// TIA Portal V17 export
// export: Created 2025-06-25T13:13:26.438801Z, ExportSetting WithDefaults, DisplayName Totally Integrated Automation Portal, DisplayVersion V17 Update 8, DisplayName TIA Portal Openness, DisplayVersion V17 Update 8, DisplayName TIA Portal Version Control Interface, DisplayVersion V17, DisplayName STEP 7 Professional, DisplayVersion V17 Update 8, DisplayName STEP 7 Safety, DisplayVersion V17 Update 6, DisplayName WinCC Advanced, DisplayVersion V17 Update 8
VAR_GLOBAL   // PLC tag table "Local_IO"
   SM1222_DO_0 AT %Q8.0 : Bool;   //    {ExternalAccessible false, ExternalVisible false, ExternalWritable false}
   SM1222_DO_1 AT %Q8.1 : Bool;   //    {ExternalAccessible false, ExternalVisible false, ExternalWritable false}
   SM1222_DO_2 AT %Q8.2 : Bool;   //    {ExternalAccessible false, ExternalVisible false, ExternalWritable false}
   SM1222_DO_3 AT %Q8.3 : Bool;   //    {ExternalAccessible false, ExternalVisible false, ExternalWritable false}
   SM1222_DO_4 AT %Q8.4 : Bool;   //    {ExternalAccessible false, ExternalVisible false, ExternalWritable false}
   SM1222_DO_5 AT %Q8.5 : Bool;   //    {ExternalAccessible false, ExternalVisible false, ExternalWritable false}
   SM1222_DO_6 AT %Q8.6 : Bool;   //    {ExternalAccessible false, ExternalVisible false, ExternalWritable false}
   SM1222_DO_7 AT %Q8.7 : Bool;   //    {ExternalAccessible false, ExternalVisible false, ExternalWritable false}
   SM531 AT %I500.0 : "stSM531_4AI";   //    {ExternalAccessible false, ExternalVisible false, ExternalWritable false}
   SM521 AT %I510.0 : "stSM521_16DI";   //    {ExternalAccessible false, ExternalVisible false, ExternalWritable false}
   SM522_I AT %I512.0 : "stSM522_32DQ_I";   //    {ExternalAccessible false, ExternalVisible false, ExternalWritable false}
   SM522_Q AT %Q512.0 : "stSM522_32DQ_Q";   //    {ExternalAccessible false, ExternalVisible false, ExternalWritable false}
END_VAR
